(* IEC 61131-3 sources: Industry-PLC-LLM/data/PLCBEAD_repo/PLCBEAD_PLCEmbed-main/PLC-BEAD/Source/GEB/GAUSS, 1 file *)

(* ---- GAUSS.ST ---- *)
FUNCTION GAUSS:REAL

	VAR_INPUT
		X :	REAL;
		U :	REAL;
		SI :	REAL;
	END_VAR

	VAR
		temp :	REAL;
		si_inv :	REAL;
	END_VAR

	temp := X - U;
	si_inv := 1.0  / SI;
	GAUSS := EXP(temp * temp * si_inv * si_inv * - 0.5) * 0.39894228 * si_inv;

END_FUNCTION

PROGRAM program0
  VAR
    X :	REAL;
	U :	REAL;
	SI :	REAL;
    LocalOUT  : REAL;
  END_VAR

  LocalOUT := GAUSS(X, U, SI);
END_PROGRAM
